{attribute 'qualified_only'}
{attribute 'strict'}
TYPE ENUM_CR_RollingConfiguration :
(
	CW2 := 0,//CW2 default
	CW1 := 1,
	DualStand := 3
);
END_TYPE

(* stored: Version 1.1.0.1, ProductVersion 3.1.4024.2
   DUT ENUM_CR_RollingConfiguration: Id {3f8408da-9f5d-4c3a-a1f6-58d2b6bab2e1} *)
